% RSLogix 500 project LIMONEIRA_2_LINE_BICARB_Modified_Sep_9_2021.RSS, saved by version 11.00.00.00 %
PROJECT "UNTITLED"    % processor: MicroLogix 1200 %

PROGRAM FILES
  LAD 2   23 rungs

DATA FILES
  O0 OUTPUT  4 elements
  I1 INPUT  4 elements
  S2 STATUS  66 elements
  B3 BINARY  1 elements
  T4 TIMER  22 elements
  C5 COUNTER  1 elements
  R6 CONTROL  1 elements
  N7 INTEGER  1 elements
  F8 FLOAT  1 elements

LADDER 2
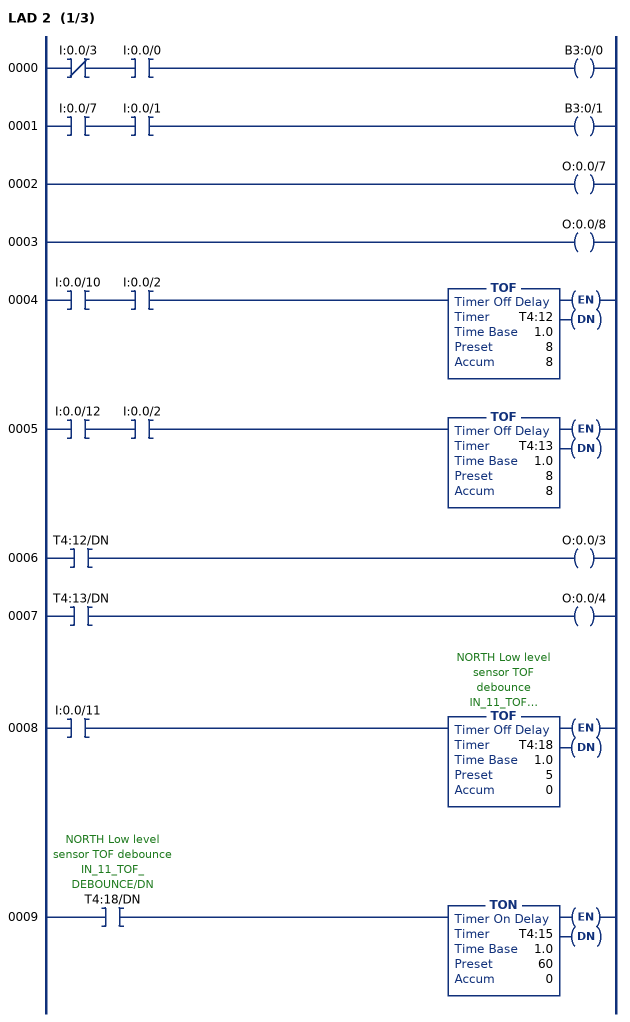
% Rung: 0 %
SOR XIO I:0.0/3 XIC I:0.0/0 OTE B3:0/0 EOR
% Rung: 1 %
SOR XIC I:0.0/7 XIC I:0.0/1 OTE B3:0/1 EOR
% Rung: 2 %
SOR OTE O:0.0/7 EOR
% Rung: 3 %
SOR OTE O:0.0/8 EOR
% Rung: 4 %
SOR XIC I:0.0/10 XIC I:0.0/2 TOF T4:12 1.0 8 8 EOR
% Rung: 5 %
SOR XIC I:0.0/12 XIC I:0.0/2 TOF T4:13 1.0 8 8 EOR
% Rung: 6 %
SOR XIC T4:12/DN OTE O:0.0/3 EOR
% Rung: 7 %
SOR XIC T4:13/DN OTE O:0.0/4 EOR
% Rung: 8 %
SOR XIC I:0.0/11 TOF T4:18 1.0 5 0 EOR
%   T4:18  IN_11_TOF_DEBOUNCE  "NORTH Low level sensor TOF debounce" %
% Rung: 9 %
SOR XIC T4:18/DN TON T4:15 1.0 60 0 EOR
%   T4:18  IN_11_TOF_DEBOUNCE  "NORTH Low level sensor TOF debounce" %

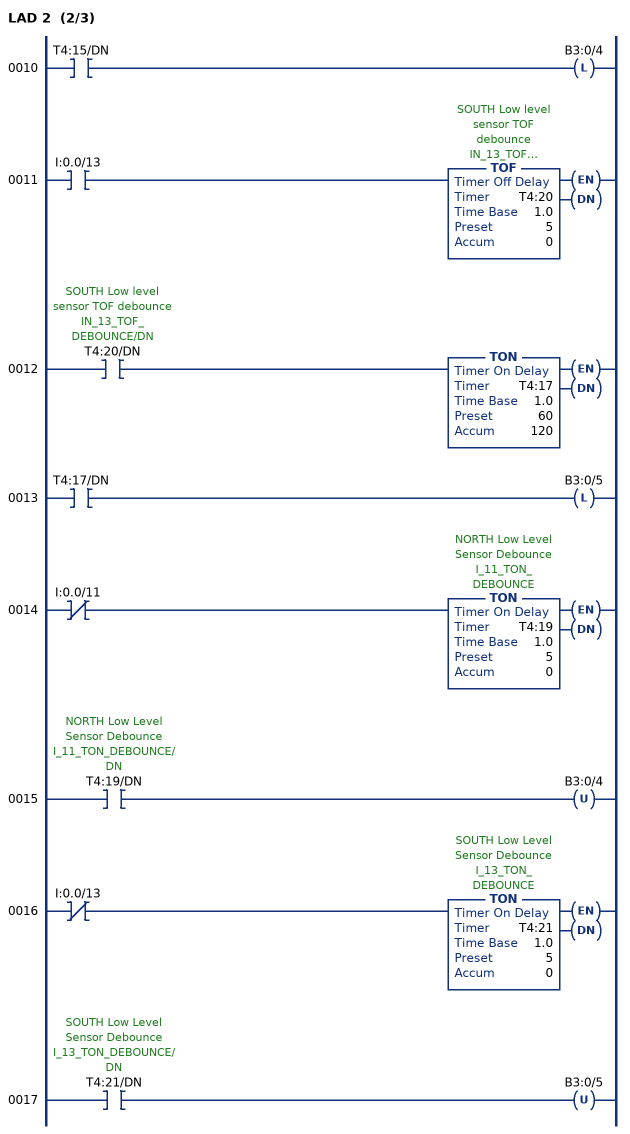
% Rung: 10 %
SOR XIC T4:15/DN OTL B3:0/4 EOR
% Rung: 11 %
SOR XIC I:0.0/13 TOF T4:20 1.0 5 0 EOR
%   T4:20  IN_13_TOF_DEBOUNCE  "SOUTH Low level sensor TOF debounce" %
% Rung: 12 %
SOR XIC T4:20/DN TON T4:17 1.0 60 120 EOR
%   T4:20  IN_13_TOF_DEBOUNCE  "SOUTH Low level sensor TOF debounce" %
% Rung: 13 %
SOR XIC T4:17/DN OTL B3:0/5 EOR
% Rung: 14 %
SOR XIO I:0.0/11 TON T4:19 1.0 5 0 EOR
%   T4:19  I_11_TON_DEBOUNCE  "NORTH Low Level Sensor Debounce" %
% Rung: 15 %
SOR XIC T4:19/DN OTU B3:0/4 EOR
%   T4:19  I_11_TON_DEBOUNCE  "NORTH Low Level Sensor Debounce" %
% Rung: 16 %
SOR XIO I:0.0/13 TON T4:21 1.0 5 0 EOR
%   T4:21  I_13_TON_DEBOUNCE  "SOUTH Low Level Sensor Debounce" %
% Rung: 17 %
SOR XIC T4:21/DN OTU B3:0/5 EOR
%   T4:21  I_13_TON_DEBOUNCE  "SOUTH Low Level Sensor Debounce" %

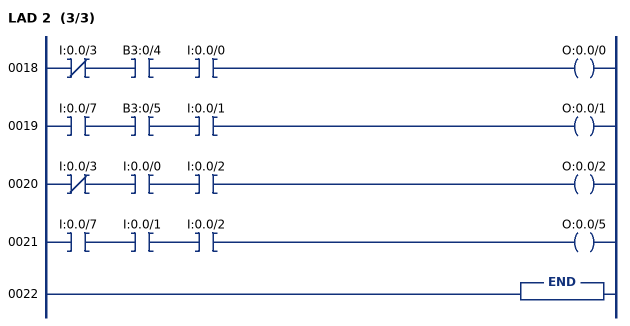
% Rung: 18 %
SOR XIO I:0.0/3 XIC B3:0/4 XIC I:0.0/0 OTE O:0.0/0 EOR
% Rung: 19 %
SOR XIC I:0.0/7 XIC B3:0/5 XIC I:0.0/1 OTE O:0.0/1 EOR
% Rung: 20 %
SOR XIO I:0.0/3 XIC I:0.0/0 XIC I:0.0/2 OTE O:0.0/2 EOR
% Rung: 21 %
SOR XIC I:0.0/7 XIC I:0.0/1 XIC I:0.0/2 OTE O:0.0/5 EOR
% Rung: 22 %
SOR END EOR

DATA TABLE (non-zero values as saved)
DATA B3
% B3:0 % 0X0033
DATA T4
% .PRE .ACC %
% T4:0 % 4 0
% T4:1 % 150 150
% T4:2 % 5 0
% T4:3 % 10 0
% T4:10 % 60 0
% T4:11 % 60 0
% T4:12 % 8 8
% T4:13 % 8 8
% T4:15 % 60 0
% T4:16 % 120 0
% T4:17 % 60 120
% T4:18 % 5 0
% T4:19 % 5 0
% T4:20 % 5 0
% T4:21 % 5 0
